// TwinCAT 3 PLC project Facade_Pattern
// ProgramVersion: 3.1.4024.0
// libraries:
//   Tc2_Standard, * (Beckhoff Automation GmbH)
//   Tc2_System, * (Beckhoff Automation GmbH)
//   Tc3_Module, * (Beckhoff Automation GmbH)
// project tree:
//   / PlcTask.TcTTO
//   POUs/ MAIN.TcPOU, XtsFacade.TcPOU
//   XTS Classes/ XtsCAGroup.TcPOU, XtsHardware.TcPOU, XtsMover.TcPOU, XtsStations.TcPOU, XtsXPU.TcPOU
// (motion and I/O tree: see PLC project simple_factory_pattern)
// real-time tasks:
//   TASK PlcTask: cycle T#10ms, priority 20, ADS port 350
//   TASK PlcTask1: cycle T#10ms, priority 21, ADS port 351
//   TASK PlcTask2: cycle T#10ms, priority 22, ADS port 352
//   TASK PlcTask3: cycle T#10ms, priority 23, ADS port 353
//   TASK PlcTask4: cycle T#10ms, priority 24, ADS port 354
//   TASK PlcTask5: cycle T#10ms, priority 25, ADS port 355
//   TASK PlcTask6: cycle T#10ms, priority 26, ADS port 356
//   TASK PlcTask7: cycle T#10ms, priority 27, ADS port 357
//   TASK PlcTask8: cycle T#10ms, priority 28, ADS port 358

CONFIGURATION Facade_Pattern
    RESOURCE PLC ON TwinCAT3
        TASK PlcTask(INTERVAL := T#10ms, PRIORITY := 28);
        PROGRAM MAIN WITH PlcTask : MAIN;
    END_RESOURCE
END_CONFIGURATION

// ---- POUs/MAIN.TcPOU
PROGRAM MAIN
VAR
	myXts : XtsFacade;
	SafetyReady: BOOL;
	XtsReady: BOOL;
END_VAR

IF SafetyReady AND NOT XtsReady THEN
	XtsReady := myXts.InitialiseXts();
END_IF

END_PROGRAM

// ---- POUs/XtsFacade.TcPOU
FUNCTION_BLOCK XtsFacade
VAR
	group : XtsCAGroup;
	hardware : XtsHardware;
	movers : ARRAY[0..10] OF XtsMover;
	stations : ARRAY[0..5] OF XtsStations;
	xpu : XtsXPU;
	i: INT;
	InitState : INT;
END_VAR

METHOD InitialiseXts : BOOL
VAR_INPUT
END_VAR
VAR
	InitCheck : BOOL;
END_VAR
CASE InitState OF
	0: 
		IF group.AddMoverToGroup() THEN
			InitState := 10;
		END_IF
	10:
		IF xpu.GetMoverInterface() THEN
			InitState := 20;
		END_IF
	20:
		InitCheck := TRUE;
		FOR i := 0 TO 5 DO
			InitCheck := InitCheck AND stations[i].InitialiseStation();
		END_FOR
		IF InitCheck THEN
			InitState := 30;
		END_IF
	30:
		IF hardware.CheckModuleVoltages() THEN
			InitState := 40;
		END_IF
	40:
		InitialiseXts := true;
END_CASE


hardware.CheckModuleVoltages();
END_METHOD

END_FUNCTION_BLOCK

// ---- XTS Classes/XtsCAGroup.TcPOU
FUNCTION_BLOCK XtsCAGroup
VAR
	Status : STRING(80);
END_VAR

METHOD AddMoverToGroup : BOOL
VAR_INPUT
END_VAR
Status := 'Movers Added To Group';
AddMoverToGroup := true;
END_METHOD

METHOD Enable : BOOL
VAR_INPUT
END_VAR
END_METHOD

END_FUNCTION_BLOCK

// ---- XTS Classes/XtsHardware.TcPOU
FUNCTION_BLOCK XtsHardware
VAR
	Status : STRING(80);
END_VAR

METHOD CheckModuleVoltages : BOOL
VAR_INPUT
END_VAR
Status := 'All Module Voltages Are OK';
CheckModuleVoltages := true;
END_METHOD

METHOD GetTrackLength : BOOL
VAR_INPUT
END_VAR
END_METHOD

END_FUNCTION_BLOCK

// ---- XTS Classes/XtsMover.TcPOU
FUNCTION_BLOCK XtsMover
VAR
END_VAR

METHOD Disable : BOOL
VAR_INPUT
END_VAR
END_METHOD

METHOD Enable : BOOL
VAR_INPUT
END_VAR
END_METHOD

METHOD MoveTo : BOOL
VAR_INPUT
END_VAR
END_METHOD

METHOD Reset : BOOL
VAR_INPUT
END_VAR
END_METHOD

END_FUNCTION_BLOCK

// ---- XTS Classes/XtsStations.TcPOU
FUNCTION_BLOCK XtsStations
VAR
	Status : STRING(80);
END_VAR

METHOD InitialiseStation : BOOL
VAR_INPUT
END_VAR
InitialiseStation := TRUE;
Status := 'Station Initialised';
END_METHOD

METHOD StationMover : BOOL
VAR_INPUT
	MoverNumber : INT;
END_VAR
END_METHOD

END_FUNCTION_BLOCK

// ---- XTS Classes/XtsXPU.TcPOU
FUNCTION_BLOCK XtsXPU
VAR
	Status : STRING(80);
END_VAR

METHOD GetMoverInterface : BOOL
VAR_INPUT
END_VAR
Status := 'Interface To XPU initialised';
GetMoverInterface := true;
END_METHOD

END_FUNCTION_BLOCK
